// TIA Portal project "Projeto Estacao Envase" (V18)
// Simulador didático de uma estação automatizada de produção e envase de garrafas, desenvolvido como recurso de apoio para uma aula técnica do SENAI.

(* hardware
DEVICE "S7-1500/ET200MP station_1"  S7-1500 station
   slot 0: "Rail_0"  Rack  6ES7 590-1***0-0AA0
   slot 1: "PLC_1"  CPU 1511C-1 PN  6ES7 511-1CK01-0AB0  V2.9
      slot 3: "CPU display_1"  6ES7591-1AA00-0AA0
      slot 32768: "PROFINET interface_1"  X1
         slot 32769: "Port_1"  X1 P1
         slot 32770: "Port_2"  X1 P2
      slot 34817: "Virtual CP interface port_1"  Virtual CP interface port  Virtual CP interface port
DEVICE "HMI_1"  KTP700 Basic PN
   slot 0: "HMI_1"  KTP700 Basic PN  6AV2 123-2GB03-0AX0  17.0.0.0
   slot 1: "HMI_RT_1"  KTP700 Basic PN  6AV2 123-2GB03-0AX0  17.0.0.0
   slot 5: "HMI_1.IE_CP_1"  PROFINET Interface  17.0.0.0
      slot 1: "PROFINET Interface_1"  PROFINET Interface
         slot 1: "Port_1"  Port
*)

// ===== PLC "PLC_1"  CPU 1511C-1 PN =====

VAR_GLOBAL   // PLC tag table "Default tag table"
   "Magazine garrafa preta recuado" AT %I10.0 : Bool;
   "Magazine garrafa preta avançado" AT %I10.1 : Bool;
   "Magazine garrafa vermelha recuado" AT %I10.2 : Bool;
   "Magazine garrafa vermelha avançado" AT %I10.3 : Bool;
   "Magazine garrafa azul recuado" AT %I10.4 : Bool;
   "Magazine garrafa azul avançado" AT %I10.5 : Bool;
   "Garrafa na posição de enchimento" AT %I10.6 : Bool;
   "Garrafa na posição de tampagem" AT %I10.7 : Bool;
   "Eixo Z recuado" AT %I11.0 : Bool;
   "Eixo X recuado" AT %I11.1 : Bool;
   "Eixo X avançado" AT %I11.2 : Bool;
   "Vácuo ligado" AT %I11.3 : Bool;
   "Avança magazine de garrafa preta" AT %Q4.0 : Bool;
   "Avança magazine de garrafa vermelha" AT %Q4.1 : Bool;
   "Avança magazine de garrafa azul" AT %Q4.2 : Bool;
   "Liga esteira" AT %Q4.3 : Bool;
   "Abre válvula de enchimento" AT %Q4.4 : Bool;
   "Desce eixo z Pick- place" AT %Q4.5 : Bool;
   "Avança eixo x Pick- place" AT %Q4.6 : Bool;
   "Liga vácuo Pick- place" AT %Q4.7 : Bool;
   "Tag_1" AT %M0.0 : Bool;
END_VAR

DATA_BLOCK "Produção_DB"   // DB1
{ S7_Optimized_Access := 'TRUE' }
VERSION : 0.1
// stored: InstanceOfName Produção
"Produção"
BEGIN
END_DATA_BLOCK

DATA_BLOCK "Magazine_DB"   // DB3
{ S7_Optimized_Access := 'TRUE' }
VERSION : 0.1
// stored: InstanceOfName Magazine
"Magazine"
BEGIN
END_DATA_BLOCK

DATA_BLOCK "Envase_DB"   // DB4
{ S7_Optimized_Access := 'TRUE' }
VERSION : 0.1
// stored: InstanceOfName Envase
"Envase"
BEGIN
END_DATA_BLOCK

DATA_BLOCK "Tampagem_DB"   // DB5
{ S7_Optimized_Access := 'TRUE' }
VERSION : 0.1
// stored: InstanceOfName Tampagem
"Tampagem"
BEGIN
END_DATA_BLOCK

// folder: System blocks/Program resources

DATA_BLOCK "IEC_Timer_0_DB"   // DB2
{ S7_Optimized_Access := 'TRUE' }
AUTHOR : Simatic
FAMILY : IEC
NAME : IEC_TMR
VERSION : 1.0
// stored: InstanceOfName IEC_TIMER
"IEC_TIMER"
BEGIN
END_DATA_BLOCK

DATA_BLOCK "IEC_Timer_0_DB_1"   // DB6
{ S7_Optimized_Access := 'TRUE' }
AUTHOR : Simatic
FAMILY : IEC
NAME : IEC_TMR
VERSION : 1.0
// stored: InstanceOfName IEC_TIMER
"IEC_TIMER"
BEGIN
END_DATA_BLOCK

DATA_BLOCK "IEC_Timer_0_DB_2"   // DB7
{ S7_Optimized_Access := 'TRUE' }
AUTHOR : Simatic
FAMILY : IEC
NAME : IEC_TMR
VERSION : 1.0
// stored: InstanceOfName IEC_TIMER
"IEC_TIMER"
BEGIN
END_DATA_BLOCK

DATA_BLOCK "IEC_Timer_0_DB_3"   // DB8
{ S7_Optimized_Access := 'TRUE' }
AUTHOR : Simatic
FAMILY : IEC
NAME : IEC_TMR
VERSION : 1.0
// stored: InstanceOfName IEC_TIMER
"IEC_TIMER"
BEGIN
END_DATA_BLOCK

DATA_BLOCK "IEC_Timer_0_DB_4"   // DB9
{ S7_Optimized_Access := 'TRUE' }
AUTHOR : Simatic
FAMILY : IEC
NAME : IEC_TMR
VERSION : 1.0
// stored: InstanceOfName IEC_TIMER
"IEC_TIMER"
BEGIN
END_DATA_BLOCK

DATA_BLOCK "IEC_Timer_0_DB_5"   // DB10
{ S7_Optimized_Access := 'TRUE' }
AUTHOR : Simatic
FAMILY : IEC
NAME : IEC_TMR
VERSION : 1.0
// stored: InstanceOfName IEC_TIMER
"IEC_TIMER"
BEGIN
END_DATA_BLOCK

DATA_BLOCK "IEC_Timer_0_DB_6"   // DB11
{ S7_Optimized_Access := 'TRUE' }
AUTHOR : Simatic
FAMILY : IEC
NAME : IEC_TMR
VERSION : 1.0
// stored: InstanceOfName IEC_TIMER
"IEC_TIMER"
BEGIN
END_DATA_BLOCK

// folder: (top level)

FUNCTION_BLOCK "Produção"   // FB1, LAD
{ S7_Optimized_Access := 'TRUE' }
VERSION : 0.1
   VAR
      passo : Int := 1;
      lp_aguardando_pedido : Bool;
      lp_start : Bool;
      lp_produção : Bool;
      produtoFinalizado : Bool;
      bt_enviarPedido : Bool;
      bt_Start : Bool;
      bt_Confirmar : Bool;
      corGarrafa : Int;
      envase : Int;
      inicioMagazine : Bool;
      finalMagazine : Bool;
      inicioEnvase : Bool;
      finalEnvase : Bool;
      inicioTampagem : Bool;
      finalTampagem : Bool;
   END_VAR
   VAR_TEMP   // added for the SCL form of the ladder/FBD networks
      _w1 : Bool;
   END_VAR
BEGIN

REGION Network 1: Passo 1 - Aguardar Pedido
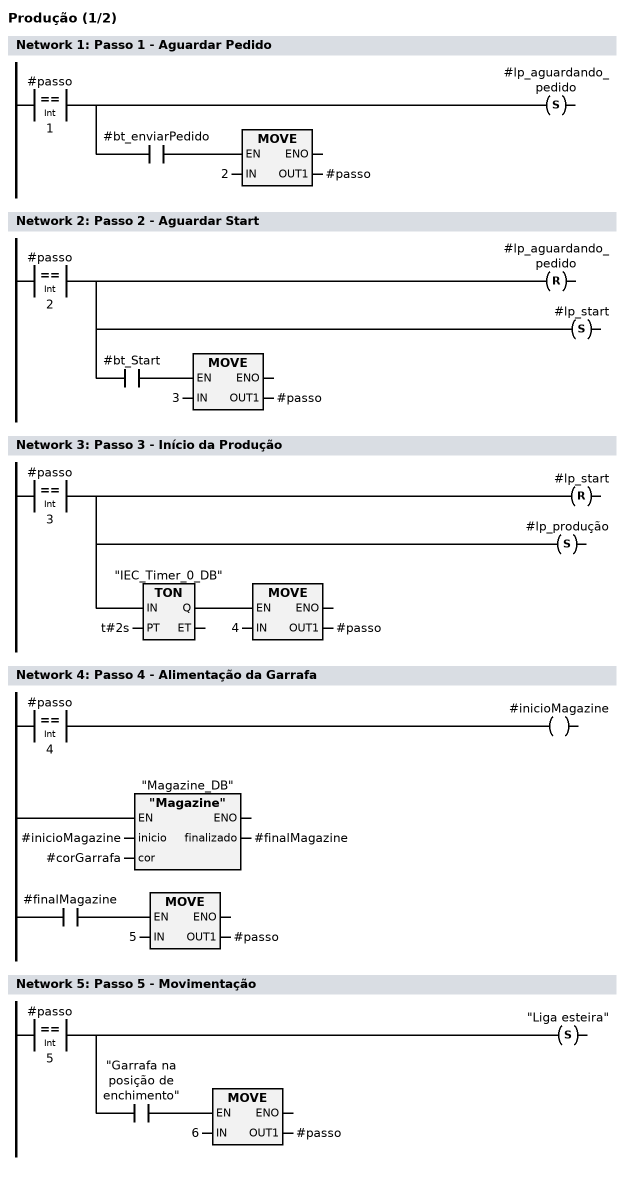
   RUNG wire#powerrail
      { S7_Templates := "SrcType := Int" } EQ_Contact(in1 := #passo, in2 := 1)
      wire#w1
      S_Coil( #lp_aguardando_pedido )
   END_RUNG
   RUNG wire#w1
      Contact( #bt_enviarPedido )
      Move(in := 2, out1 => #passo)
   END_RUNG
   // the same network as SCL:
   #_w1 := #passo = 1;
   IF #_w1 THEN #lp_aguardando_pedido := TRUE; END_IF;
   IF #_w1 AND #bt_enviarPedido THEN #passo := 2; END_IF;
END_REGION

REGION Network 2: Passo 2 - Aguardar Start
   RUNG wire#powerrail
      { S7_Templates := "SrcType := Int" } EQ_Contact(in1 := #passo, in2 := 2)
      wire#w1
      R_Coil( #lp_aguardando_pedido )
   END_RUNG
   RUNG wire#w1
      S_Coil( #lp_start )
   END_RUNG
   RUNG wire#w1
      Contact( #bt_Start )
      Move(in := 3, out1 => #passo)
   END_RUNG
   // the same network as SCL:
   #_w1 := #passo = 2;
   IF #_w1 THEN
       #lp_aguardando_pedido := FALSE;
       #lp_start := TRUE;
   END_IF;
   IF #_w1 AND #bt_Start THEN #passo := 3; END_IF;
END_REGION

REGION Network 3: Passo 3 - Início da Produção
   #_w1 := #passo = 3;
   IF #_w1 THEN
       #lp_start := FALSE;
       #lp_produção := TRUE;
   END_IF;
   "IEC_Timer_0_DB".TON(IN := #_w1, PT := t#2s);
   IF "IEC_Timer_0_DB".Q THEN #passo := 4; END_IF;
END_REGION

REGION Network 4: Passo 4 - Alimentação da Garrafa
   RUNG wire#powerrail
      { S7_Templates := "SrcType := Int" } EQ_Contact(in1 := #passo, in2 := 4)
      Coil( #inicioMagazine )
   END_RUNG
   RUNG wire#powerrail
      "Magazine_DB"(inicio := #inicioMagazine, cor := #corGarrafa, finalizado => #finalMagazine)
   END_RUNG
   RUNG wire#powerrail
      Contact( #finalMagazine )
      Move(in := 5, out1 => #passo)
   END_RUNG
   // the same network as SCL:
   #inicioMagazine := #passo = 4;
   "Magazine_DB"(inicio := #inicioMagazine, cor := #corGarrafa, finalizado => #finalMagazine);   // "Magazine"
   IF #finalMagazine THEN #passo := 5; END_IF;
END_REGION

REGION Network 5: Passo 5 - Movimentação
   RUNG wire#powerrail
      { S7_Templates := "SrcType := Int" } EQ_Contact(in1 := #passo, in2 := 5)
      wire#w1
      S_Coil( "Liga esteira" )
   END_RUNG
   RUNG wire#w1
      Contact( "Garrafa na posição de enchimento" )
      Move(in := 6, out1 => #passo)
   END_RUNG
   // the same network as SCL:
   #_w1 := #passo = 5;
   IF #_w1 THEN "Liga esteira" := TRUE; END_IF;
   IF #_w1 AND "Garrafa na posição de enchimento" THEN #passo := 6; END_IF;
END_REGION

REGION Network 6: Passo 6 - Enchimento/Envase
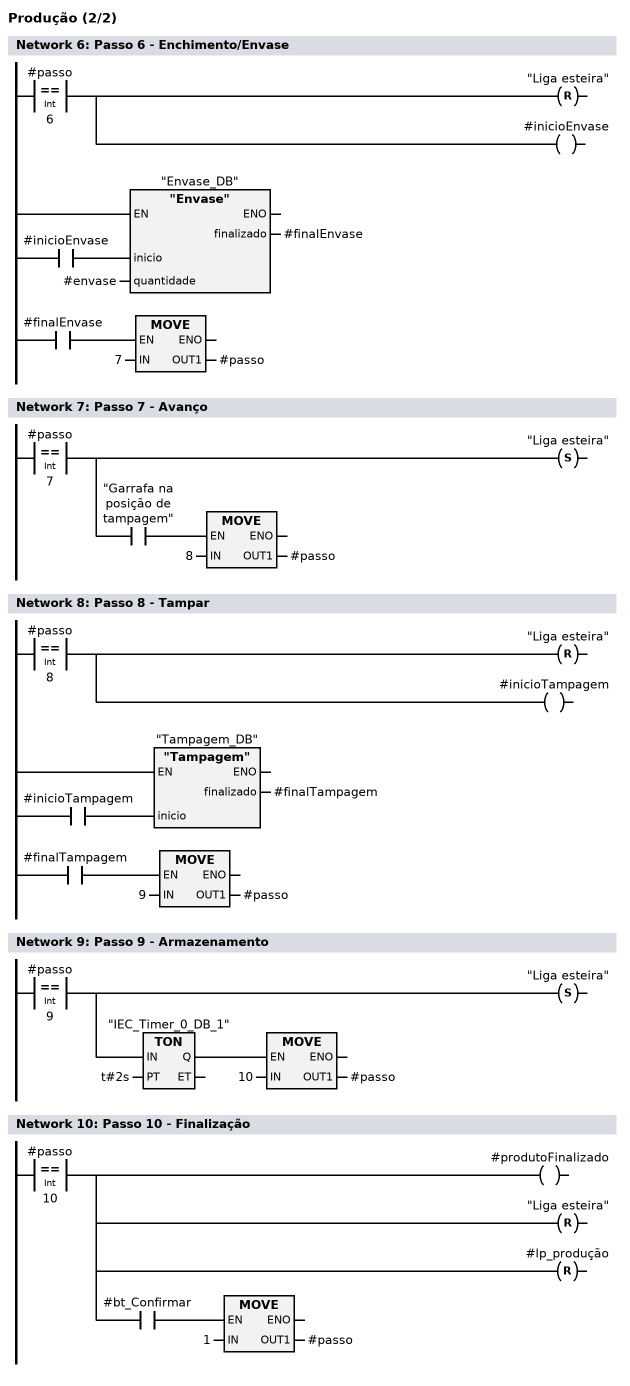
   RUNG wire#powerrail
      { S7_Templates := "SrcType := Int" } EQ_Contact(in1 := #passo, in2 := 6)
      wire#w1
      R_Coil( "Liga esteira" )
   END_RUNG
   RUNG wire#w1
      Coil( #inicioEnvase )
   END_RUNG
   RUNG wire#powerrail
      "Envase_DB"(inicio := wire#w2, quantidade := #envase, finalizado => #finalEnvase)
   END_RUNG
   RUNG wire#powerrail
      Contact( #inicioEnvase )
   END_RUNG wire#w2
   RUNG wire#powerrail
      Contact( #finalEnvase )
      Move(in := 7, out1 => #passo)
   END_RUNG
   // the same network as SCL:
   #_w1 := #passo = 6;
   IF #_w1 THEN "Liga esteira" := FALSE; END_IF;
   #inicioEnvase := #_w1;
   "Envase_DB"(inicio := #inicioEnvase, quantidade := #envase, finalizado => #finalEnvase);   // "Envase"
   IF #finalEnvase THEN #passo := 7; END_IF;
END_REGION

REGION Network 7: Passo 7 - Avanço
   RUNG wire#powerrail
      { S7_Templates := "SrcType := Int" } EQ_Contact(in1 := #passo, in2 := 7)
      wire#w1
      S_Coil( "Liga esteira" )
   END_RUNG
   RUNG wire#w1
      Contact( "Garrafa na posição de tampagem" )
      Move(in := 8, out1 => #passo)
   END_RUNG
   // the same network as SCL:
   #_w1 := #passo = 7;
   IF #_w1 THEN "Liga esteira" := TRUE; END_IF;
   IF #_w1 AND "Garrafa na posição de tampagem" THEN #passo := 8; END_IF;
END_REGION

REGION Network 8: Passo 8 - Tampar
   RUNG wire#powerrail
      { S7_Templates := "SrcType := Int" } EQ_Contact(in1 := #passo, in2 := 8)
      wire#w1
      R_Coil( "Liga esteira" )
   END_RUNG
   RUNG wire#w1
      Coil( #inicioTampagem )
   END_RUNG
   RUNG wire#powerrail
      "Tampagem_DB"(inicio := wire#w2, finalizado => #finalTampagem)
   END_RUNG
   RUNG wire#powerrail
      Contact( #inicioTampagem )
   END_RUNG wire#w2
   RUNG wire#powerrail
      Contact( #finalTampagem )
      Move(in := 9, out1 => #passo)
   END_RUNG
   // the same network as SCL:
   #_w1 := #passo = 8;
   IF #_w1 THEN "Liga esteira" := FALSE; END_IF;
   #inicioTampagem := #_w1;
   "Tampagem_DB"(inicio := #inicioTampagem, finalizado => #finalTampagem);   // "Tampagem"
   IF #finalTampagem THEN #passo := 9; END_IF;
END_REGION

REGION Network 9: Passo 9 - Armazenamento
   #_w1 := #passo = 9;
   IF #_w1 THEN "Liga esteira" := TRUE; END_IF;
   "IEC_Timer_0_DB_1".TON(IN := #_w1, PT := t#2s);
   IF "IEC_Timer_0_DB_1".Q THEN #passo := 10; END_IF;
END_REGION

REGION Network 10: Passo 10 - Finalização
   RUNG wire#powerrail
      { S7_Templates := "SrcType := Int" } EQ_Contact(in1 := #passo, in2 := 10)
      wire#w1
      Coil( #produtoFinalizado )
   END_RUNG
   RUNG wire#w1
      R_Coil( "Liga esteira" )
   END_RUNG
   RUNG wire#w1
      R_Coil( #lp_produção )
   END_RUNG
   RUNG wire#w1
      Contact( #bt_Confirmar )
      Move(in := 1, out1 => #passo)
   END_RUNG
   // the same network as SCL:
   #produtoFinalizado := #passo = 10;
   IF #produtoFinalizado THEN
       "Liga esteira" := FALSE;
       #lp_produção := FALSE;
   END_IF;
   IF #produtoFinalizado AND #bt_Confirmar THEN #passo := 1; END_IF;
END_REGION
END_FUNCTION_BLOCK

FUNCTION_BLOCK "Magazine"   // FB2, LAD
{ S7_Optimized_Access := 'TRUE' }
VERSION : 0.1
   VAR_INPUT
      inicio : Bool;
      cor : Int;
   END_VAR
   VAR_OUTPUT
      finalizado : Bool;
   END_VAR
   VAR
      passo : Int := 1;
   END_VAR
   VAR_TEMP   // added for the SCL form of the ladder/FBD networks
      _w1 : Bool;
      _w2 : Bool;
      _w3 : Bool;
      _w4 : Bool;
   END_VAR
BEGIN

REGION Network 1: Avançar/Alimentar
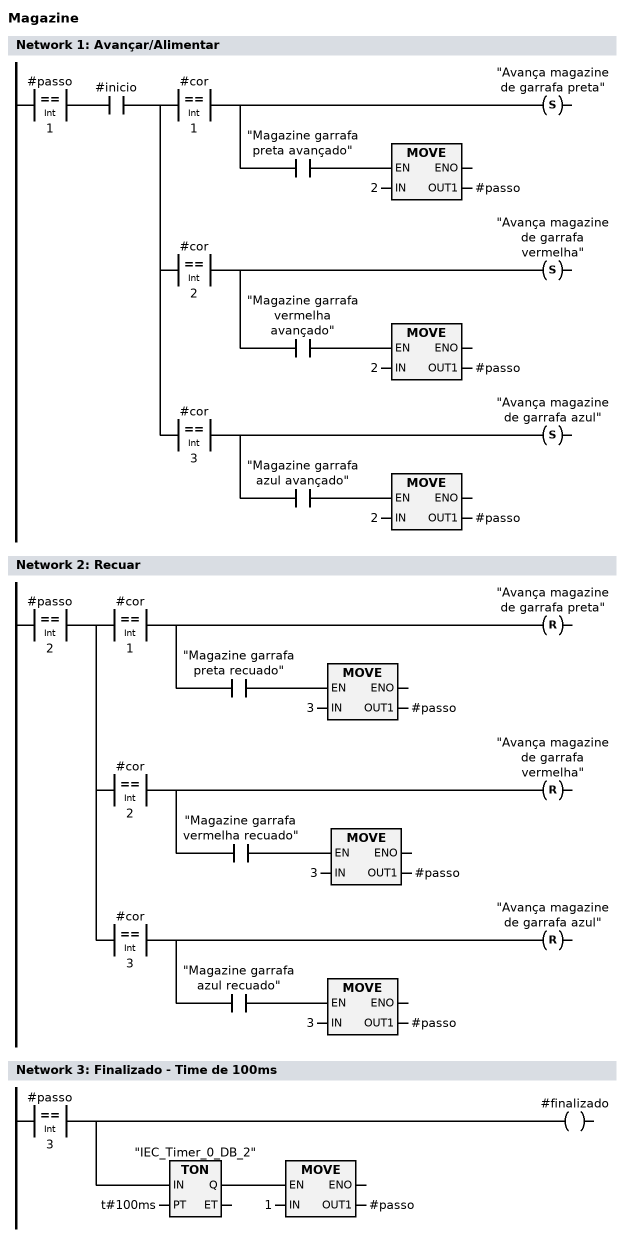
   RUNG wire#powerrail
      { S7_Templates := "SrcType := Int" } EQ_Contact(in1 := #passo, in2 := 1)
      Contact( #inicio )
      wire#w1
      { S7_Templates := "SrcType := Int" } EQ_Contact(in1 := #cor, in2 := 1)
      wire#w2
      S_Coil( "Avança magazine de garrafa preta" )
   END_RUNG
   RUNG wire#w2
      Contact( "Magazine garrafa preta avançado" )
      Move(in := 2, out1 => #passo)
   END_RUNG
   RUNG wire#w1
      { S7_Templates := "SrcType := Int" } EQ_Contact(in1 := #cor, in2 := 2)
      wire#w3
      S_Coil( "Avança magazine de garrafa vermelha" )
   END_RUNG
   RUNG wire#w3
      Contact( "Magazine garrafa vermelha avançado" )
      Move(in := 2, out1 => #passo)
   END_RUNG
   RUNG wire#w1
      { S7_Templates := "SrcType := Int" } EQ_Contact(in1 := #cor, in2 := 3)
      wire#w4
      S_Coil( "Avança magazine de garrafa azul" )
   END_RUNG
   RUNG wire#w4
      Contact( "Magazine garrafa azul avançado" )
      Move(in := 2, out1 => #passo)
   END_RUNG
   // the same network as SCL:
   #_w1 := (#passo = 1) AND #inicio;
   #_w2 := #_w1 AND (#cor = 1);
   IF #_w2 THEN "Avança magazine de garrafa preta" := TRUE; END_IF;
   IF #_w2 AND "Magazine garrafa preta avançado" THEN #passo := 2; END_IF;
   #_w3 := #_w1 AND (#cor = 2);
   IF #_w3 THEN "Avança magazine de garrafa vermelha" := TRUE; END_IF;
   IF #_w3 AND "Magazine garrafa vermelha avançado" THEN #passo := 2; END_IF;
   #_w4 := #_w1 AND (#cor = 3);
   IF #_w4 THEN "Avança magazine de garrafa azul" := TRUE; END_IF;
   IF #_w4 AND "Magazine garrafa azul avançado" THEN #passo := 2; END_IF;
END_REGION

REGION Network 2: Recuar
   RUNG wire#powerrail
      { S7_Templates := "SrcType := Int" } EQ_Contact(in1 := #passo, in2 := 2)
      wire#w1
      { S7_Templates := "SrcType := Int" } EQ_Contact(in1 := #cor, in2 := 1)
      wire#w2
      R_Coil( "Avança magazine de garrafa preta" )
   END_RUNG
   RUNG wire#w2
      Contact( "Magazine garrafa preta recuado" )
      Move(in := 3, out1 => #passo)
   END_RUNG
   RUNG wire#w1
      { S7_Templates := "SrcType := Int" } EQ_Contact(in1 := #cor, in2 := 2)
      wire#w3
      R_Coil( "Avança magazine de garrafa vermelha" )
   END_RUNG
   RUNG wire#w3
      Contact( "Magazine garrafa vermelha recuado" )
      Move(in := 3, out1 => #passo)
   END_RUNG
   RUNG wire#w1
      { S7_Templates := "SrcType := Int" } EQ_Contact(in1 := #cor, in2 := 3)
      wire#w4
      R_Coil( "Avança magazine de garrafa azul" )
   END_RUNG
   RUNG wire#w4
      Contact( "Magazine garrafa azul recuado" )
      Move(in := 3, out1 => #passo)
   END_RUNG
   // the same network as SCL:
   #_w1 := #passo = 2;
   #_w2 := #_w1 AND (#cor = 1);
   IF #_w2 THEN "Avança magazine de garrafa preta" := FALSE; END_IF;
   IF #_w2 AND "Magazine garrafa preta recuado" THEN #passo := 3; END_IF;
   #_w3 := #_w1 AND (#cor = 2);
   IF #_w3 THEN "Avança magazine de garrafa vermelha" := FALSE; END_IF;
   IF #_w3 AND "Magazine garrafa vermelha recuado" THEN #passo := 3; END_IF;
   #_w4 := #_w1 AND (#cor = 3);
   IF #_w4 THEN "Avança magazine de garrafa azul" := FALSE; END_IF;
   IF #_w4 AND "Magazine garrafa azul recuado" THEN #passo := 3; END_IF;
END_REGION

REGION Network 3: Finalizado - Time de 100ms
   #finalizado := #passo = 3;
   "IEC_Timer_0_DB_2".TON(IN := #finalizado, PT := t#100ms);
   IF "IEC_Timer_0_DB_2".Q THEN #passo := 1; END_IF;
END_REGION
END_FUNCTION_BLOCK

FUNCTION_BLOCK "Envase"   // FB3, LAD
{ S7_Optimized_Access := 'TRUE' }
VERSION : 0.1
   VAR_INPUT
      inicio : Bool;
      quantidade : Int;
   END_VAR
   VAR_OUTPUT
      finalizado : Bool;
   END_VAR
   VAR
      envaseAtual : Int;
      reset_time : Bool;
   END_VAR
   VAR_TEMP   // added for the SCL form of the ladder/FBD networks
      _w1 : Bool;
   END_VAR
BEGIN

REGION Network 1
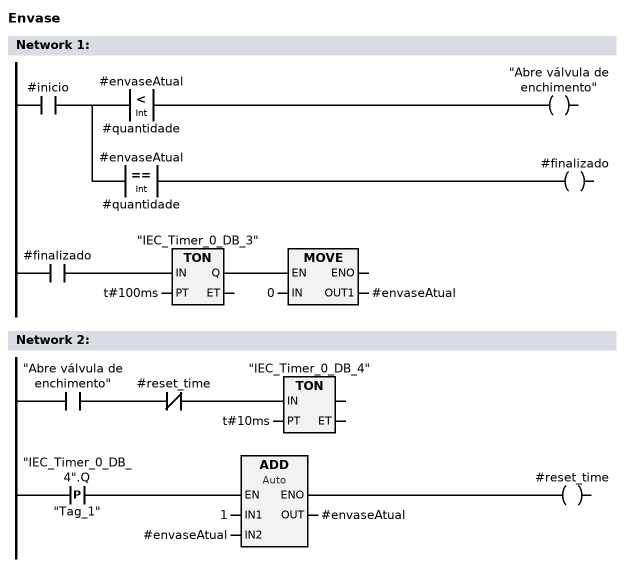
   "Abre válvula de enchimento" := #inicio AND (#envaseAtual < #quantidade);
   #finalizado := #inicio AND (#envaseAtual = #quantidade);
   "IEC_Timer_0_DB_3".TON(IN := #finalizado, PT := t#100ms);
   IF "IEC_Timer_0_DB_3".Q THEN #envaseAtual := 0; END_IF;
END_REGION

REGION Network 2
   "IEC_Timer_0_DB_4".TON(IN := "Abre válvula de enchimento" AND NOT #reset_time, PT := t#10ms);
   #_w1 := "IEC_Timer_0_DB_4".Q AND NOT "Tag_1";   // rising edge of "IEC_Timer_0_DB_4".Q
   "Tag_1" := "IEC_Timer_0_DB_4".Q;
   IF #_w1 THEN #envaseAtual := 1 + #envaseAtual; END_IF;
   #reset_time := #_w1;
END_REGION
END_FUNCTION_BLOCK

FUNCTION_BLOCK "Tampagem"   // FB4, LAD
{ S7_Optimized_Access := 'TRUE' }
VERSION : 0.1
   VAR_INPUT
      inicio : Bool;
   END_VAR
   VAR_OUTPUT
      finalizado : Bool;
   END_VAR
   VAR
      passo : Int := 1;
   END_VAR
   VAR_TEMP   // added for the SCL form of the ladder/FBD networks
      _w1 : Bool;
   END_VAR
BEGIN

REGION Network 1: Recuar Eixo X
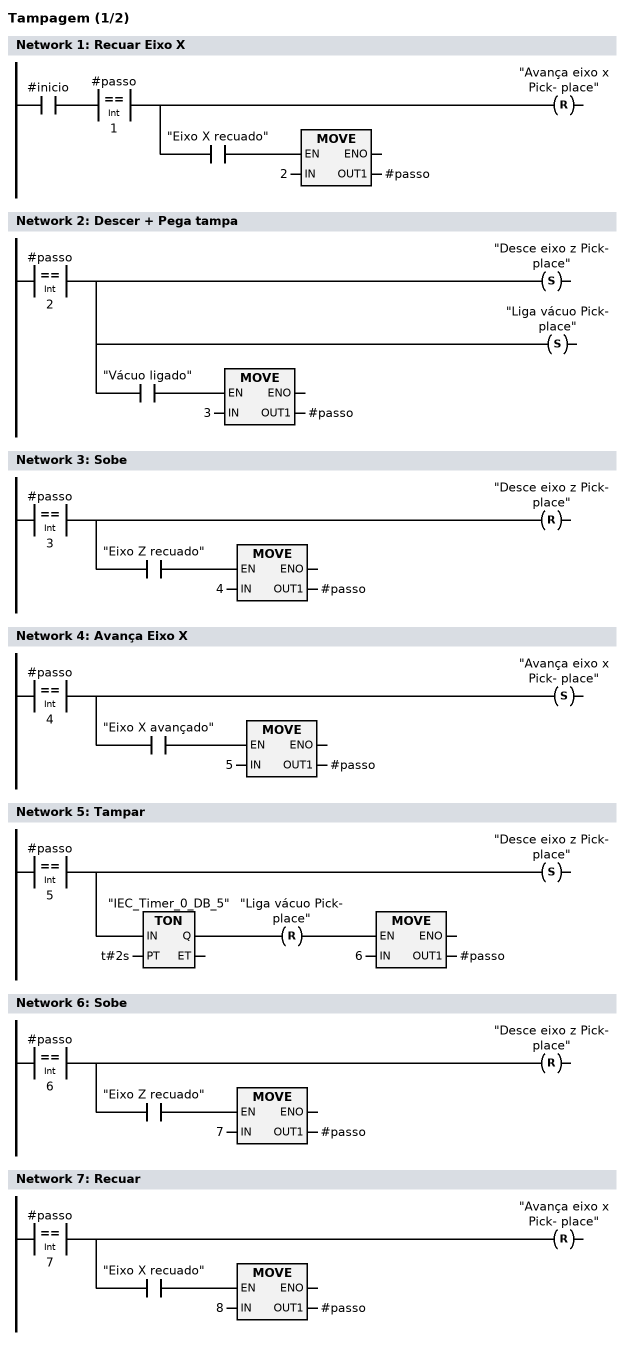
   RUNG wire#powerrail
      Contact( #inicio )
      { S7_Templates := "SrcType := Int" } EQ_Contact(in1 := #passo, in2 := 1)
      wire#w1
      R_Coil( "Avança eixo x Pick- place" )
   END_RUNG
   RUNG wire#w1
      Contact( "Eixo X recuado" )
      Move(in := 2, out1 => #passo)
   END_RUNG
   // the same network as SCL:
   #_w1 := #inicio AND (#passo = 1);
   IF #_w1 THEN "Avança eixo x Pick- place" := FALSE; END_IF;
   IF #_w1 AND "Eixo X recuado" THEN #passo := 2; END_IF;
END_REGION

REGION Network 2: Descer + Pega tampa
   RUNG wire#powerrail
      { S7_Templates := "SrcType := Int" } EQ_Contact(in1 := #passo, in2 := 2)
      wire#w1
      S_Coil( "Desce eixo z Pick- place" )
   END_RUNG
   RUNG wire#w1
      S_Coil( "Liga vácuo Pick- place" )
   END_RUNG
   RUNG wire#w1
      Contact( "Vácuo ligado" )
      Move(in := 3, out1 => #passo)
   END_RUNG
   // the same network as SCL:
   #_w1 := #passo = 2;
   IF #_w1 THEN
       "Desce eixo z Pick- place" := TRUE;
       "Liga vácuo Pick- place" := TRUE;
   END_IF;
   IF #_w1 AND "Vácuo ligado" THEN #passo := 3; END_IF;
END_REGION

REGION Network 3: Sobe
   RUNG wire#powerrail
      { S7_Templates := "SrcType := Int" } EQ_Contact(in1 := #passo, in2 := 3)
      wire#w1
      R_Coil( "Desce eixo z Pick- place" )
   END_RUNG
   RUNG wire#w1
      Contact( "Eixo Z recuado" )
      Move(in := 4, out1 => #passo)
   END_RUNG
   // the same network as SCL:
   #_w1 := #passo = 3;
   IF #_w1 THEN "Desce eixo z Pick- place" := FALSE; END_IF;
   IF #_w1 AND "Eixo Z recuado" THEN #passo := 4; END_IF;
END_REGION

REGION Network 4: Avança Eixo X
   RUNG wire#powerrail
      { S7_Templates := "SrcType := Int" } EQ_Contact(in1 := #passo, in2 := 4)
      wire#w1
      S_Coil( "Avança eixo x Pick- place" )
   END_RUNG
   RUNG wire#w1
      Contact( "Eixo X avançado" )
      Move(in := 5, out1 => #passo)
   END_RUNG
   // the same network as SCL:
   #_w1 := #passo = 4;
   IF #_w1 THEN "Avança eixo x Pick- place" := TRUE; END_IF;
   IF #_w1 AND "Eixo X avançado" THEN #passo := 5; END_IF;
END_REGION

REGION Network 5: Tampar
   #_w1 := #passo = 5;
   IF #_w1 THEN "Desce eixo z Pick- place" := TRUE; END_IF;
   "IEC_Timer_0_DB_5".TON(IN := #_w1, PT := t#2s);
   IF "IEC_Timer_0_DB_5".Q THEN
       "Liga vácuo Pick- place" := FALSE;
       #passo := 6;
   END_IF;
END_REGION

REGION Network 6: Sobe
   RUNG wire#powerrail
      { S7_Templates := "SrcType := Int" } EQ_Contact(in1 := #passo, in2 := 6)
      wire#w1
      R_Coil( "Desce eixo z Pick- place" )
   END_RUNG
   RUNG wire#w1
      Contact( "Eixo Z recuado" )
      Move(in := 7, out1 => #passo)
   END_RUNG
   // the same network as SCL:
   #_w1 := #passo = 6;
   IF #_w1 THEN "Desce eixo z Pick- place" := FALSE; END_IF;
   IF #_w1 AND "Eixo Z recuado" THEN #passo := 7; END_IF;
END_REGION

REGION Network 7: Recuar
   RUNG wire#powerrail
      { S7_Templates := "SrcType := Int" } EQ_Contact(in1 := #passo, in2 := 7)
      wire#w1
      R_Coil( "Avança eixo x Pick- place" )
   END_RUNG
   RUNG wire#w1
      Contact( "Eixo X recuado" )
      Move(in := 8, out1 => #passo)
   END_RUNG
   // the same network as SCL:
   #_w1 := #passo = 7;
   IF #_w1 THEN "Avança eixo x Pick- place" := FALSE; END_IF;
   IF #_w1 AND "Eixo X recuado" THEN #passo := 8; END_IF;
END_REGION

REGION Network 8: Finalizar
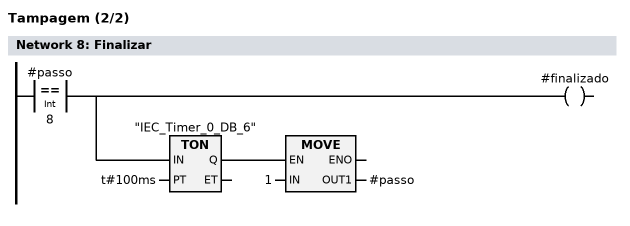
   #finalizado := #passo = 8;
   "IEC_Timer_0_DB_6".TON(IN := #finalizado, PT := t#100ms);
   IF "IEC_Timer_0_DB_6".Q THEN #passo := 1; END_IF;
END_REGION
END_FUNCTION_BLOCK

ORGANIZATION_BLOCK "Main"   // OB1, LAD, ProgramCycle
TITLE = "Main Program Sweep (Cycle)"
{ S7_Optimized_Access := 'TRUE' }
VERSION : 0.1
   VAR_INPUT
      Initial_Call : Bool;   // Initial call of this OB
      Remanence : Bool;   // =True, if remanent data are available
   END_VAR
BEGIN

REGION Network 1
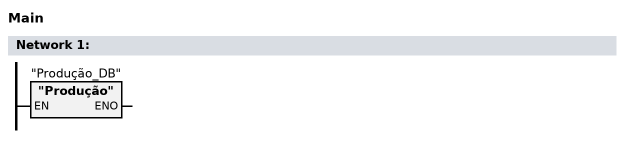
   RUNG wire#powerrail
      "Produção_DB"()
   END_RUNG
   // the same network as SCL:
   "Produção_DB"();   // "Produção"
END_REGION
END_ORGANIZATION_BLOCK

(* ===== HMI "HMI_RT_1" =====
system functions are stored by id; their names below are inferred from use
connection "HMI_Connection_1": ETHERNET, SMART_S7_1500_OMS

HMI tags "Default tag table"
   "AguardandoPedido" : Bool = PLC Produção_DB.lp_aguardando_pedido AT %DB1.DBX0.0, 100 ms
   "AguardandoStart" : Bool = PLC Produção_DB.lp_start AT %DB1.DBX0.0, 100 ms
   "EmProducao" : Bool = PLC Produção_DB.lp_produção AT %DB1.DBX0.0, 100 ms
   "ProdutoFinalizado" : Bool = PLC Produção_DB.produtoFinalizado AT %DB1.DBX0.0, 100 ms
   "bt_ConfirmaPedido" : Bool = PLC Produção_DB.bt_Confirmar AT %DB1.DBX0.0, 100 ms
   "bt_Start" : Bool = PLC Produção_DB.bt_Start AT %DB1.DBX0.0, 100 ms
   "bt_EnviaPedido" : Bool = PLC Produção_DB.bt_enviarPedido AT %DB1.DBX0.0, 100 ms
   "CorGarrafa" : Int = PLC Produção_DB.corGarrafa AT %DB1.DBW0, 100 ms
   "Envase" : Int = PLC Produção_DB.envase AT %DB1.DBW0, 100 ms
   "EnvaseAtual" : Int = PLC Envase_DB.envaseAtual AT %DB1.DBW0, 100 ms

Template "Template_1" 800x480
   Button "Exit" at 714,429 size 71x50; TextOff 'Exit'; PictureOff "ExitRuntime_KTP700_Basic_PN_TR"; PictureOn "ExitRuntime_KTP700_Basic_PN_TR"
      on Release: StopRuntime(0)
   Button "Template_Button" at 614,429 size 71x50; TextOff 'Text'
   Button "Template_Button_1" at 514,429 size 71x50; TextOff 'Text'
   Button "Template_Button_2" at 414,429 size 71x50; TextOff 'Text'
   Button "Template_Button_3" at 314,429 size 71x50; TextOff 'Text'
   Button "Template_Button_4" at 214,429 size 71x50; TextOff 'Text'
   Button "Template_Button_5" at 114,429 size 71x50; TextOff 'Text'
   Button "Start screen" at 14,429 size 71x50; TextOff 'Start screen'; PictureOff "NavigateHome_KTP700_Basic_PN_TR"; PictureOn "NavigateHome_KTP700_Basic_PN_TR"
      on Release: ActivateScreen("Root screen", 0)
   SymbolicIOField "Symbolic_IO_Field_Screen" at 93,9 size 600x33; TextOff '0'; TextOn '1'; TextList "TextList_ScreenNames"
      ProcessValue <- "AguardandoPedido"
      on Change: ActivateScreenByNumber("AguardandoPedido", 0)
   DateTimeField "HmiScreenItemData" at 695,25 size 105x25
   DateTimeField "HmiScreenItemData_1" at 695,0 size 105x25
   GraphicView "Logo" at 0,0 size 91x51; Picture "Logo of HMI_1"

screen "Root screen" 800x480, template "Template_1"
   on GenerateScreen: SetTag("AguardandoPedido", 1)
   Button "Button_1" at 88,209 size 174x32; TextOff 'Enviar Pedido'
      on Press: SetBit("bt_EnviaPedido")
      on Release: ResetBit("bt_EnviaPedido")
   Button "Button_2" at 307,207 size 174x32; TextOff 'Start'
      on Press: SetBit("bt_Start")
      on Release: ResetBit("bt_Start")
   Button "Button_3" at 526,205 size 174x32; TextOff 'Confirmar Produção'
      on Press: SetBit("bt_ConfirmaPedido")
      on Release: ResetBit("bt_ConfirmaPedido")
   TextField "Text field_1" at 93,52 size 165x23; Text 'Aguardando Pedido'
   TextField "Text field_2" at 319,51 size 150x23; Text 'Aguardando Start'
   TextField "Text field_3" at 557,51 size 111x23; Text 'Em Produção'
   Circle "Circle_1" at 137,94 size 77x77
      Appearance <- "AguardandoPedido"
   Circle "Circle_2" at 356,91 size 77x77
      Appearance <- "AguardandoStart"
   Circle "Circle_3" at 574,91 size 77x77
      Appearance <- "EmProducao"
   TextField "Text field_4" at 105,391 size 345x39; Text 'PRODUTO FINALIZADO'
      Visibility <- "ProdutoFinalizado"
   TextField "Text field_5" at 101,267 size 139x32; Text 'Cor Garrafa'
   TextField "Text field_6" at 348,267 size 87x32; Text 'Envase'
   SymbolicIOField "Symbolic I/O field_1" at 110,316 size 120x48; TextOff '0'; TextOn '1'; TextList "TextList_ScreenNames"
      ProcessValue <- "CorGarrafa"
   IOField "I/O field_1" at 330,316 size 120x48; FormatPattern 9999
      ProcessValue <- "Envase"
   TextField "Text field_7" at 557,242 size 111x23; Text 'Envase Atual'
   Bar "Bar_1" at 548,279 size 129x174; MinimumValue 0; MaximumValue 1000
      ProcessValue <- "EnvaseAtual"
*)